TYPE T_JUMO_CTRL EXTENDS T_RS_BASE_CTRL:
STRUCT
	nSlaveID:	BYTE 	:= 1;						// Modbus Slave ID, 1..247
	nCmdType:	DINT	:= E_MODBUS_CMD_TYPE.READ;	// Command type; 0-Read, 1-Write
	nRegister:	DINT;								// Command register
	nWords:		DINT	:= 1;						// Number of words
	nValue:		DINT;								// Parameter value
END_STRUCT
END_TYPE

(* stored: Version 1.1.0.1, ProductVersion 3.1.4022.16
   DUT T_JUMO_CTRL: Id {7339fb85-855d-4ffd-87c1-4f959e5e3e3c} *)
